PROGRAM Simulation
VAR
END_VAR

VAL.bValve_A_AtHomeSensor:=VAL.bValve_A_HomeCmd;
VAL.bValve_A_AtWorkSensor:=VAL.bValve_A_WorkCmd;

VAL.bValve_B_AtHomeSensor:=VAL.bValve_B_HomeCmd;
VAL.bValve_B_AtWorkSensor:=VAL.bValve_B_WorkCmd;

VAL.bValve_C_AtHomeSensor:=VAL.bValve_C_HomeCmd;
VAL.bValve_C_AtWorkSensor:=VAL.bValve_C_WorkCmd;

VAL.bValve_D_AtHomeSensor:=VAL.bValve_D_HomeCmd;
VAL.bValve_D_AtWorkSensor:=VAL.bValve_D_WorkCmd;

END_PROGRAM

(* stored: Version 1.1.0.1, ProductVersion 3.1.4024.12
   POU Simulation: Id {af3556ba-86fc-4643-ae50-def7bac0638d}, SpecialFunc None *)
